FUNCTION_BLOCK "LER_SoftCam_Interface"
{ S7_Optimized_Access := 'TRUE' ; Published := 'TRUE' }
VERSION : 0.1
   VAR_INPUT
      axis64PosInterface : "LBC_typeAxis64PosInterface";
   END_VAR

   VAR_IN_OUT
      softCam : "LER_typeSoftCamInterface";
   END_VAR

   VAR_TEMP
      tempLoopCount : Int;
   END_VAR


BEGIN
END_FUNCTION_BLOCK

